(* CoDeSys 2.3.9.42 project: komp.pro *)
(* Libraries: Standard.lib 2.12.10 17:48:34, SYSLIBCALLBACK.LIB 2.12.10 17:48:32 *)

(* PLC configuration (modules and I/O channels)
0750-1405 16 DI 24V DC 3.0ms [Type_1_16_Channels] node 0, in %IB24 out %QB0 {INTTypePAAssignment = PLC; INTTypeModule = plugged}
  AT %IX12.0 [BOOLOnX_I] Ch_1 Digital input
  AT %IX12.1 [BOOLOnX_I] Ch_2 Digital input
  AT %IX12.2 [BOOLOnX_I] Ch_3 Digital input
  AT %IX12.3 [BOOLOnX_I] Ch_4 Digital input
  AT %IX12.4 [BOOLOnX_I] Ch_5 Digital input
  AT %IX12.5 [BOOLOnX_I] Ch_6 Digital input
  AT %IX12.6 [BOOLOnX_I] Ch_7 Digital input
  AT %IX12.7 [BOOLOnX_I] Ch_8 Digital input
  AT %IX12.8 [BOOLOnX_I] Ch_9 Digital input
  AT %IX12.9 [BOOLOnX_I] Ch_10 Digital input
  AT %IX12.10 [BOOLOnX_I] Ch_11 Digital input
  AT %IX12.11 [BOOLOnX_I] Ch_12 Digital input
  AT %IX12.12 [BOOLOnX_I] Ch_13 Digital input
  AT %IX12.13 [BOOLOnX_I] Ch_14 Digital input
  AT %IX12.14 [BOOLOnX_I] Ch_15 Digital input
  AT %IX12.15 [BOOLOnX_I] Ch_16 Digital input
0750-1405 16 DI 24V DC 3.0ms [Type_1_16_Channels] node 0, in %IB24 out %QB0 {INTTypePAAssignment = PLC; INTTypeModule = plugged}
  AT %IX13.0 [BOOLOnX_I] Ch_1 Digital input
  AT %IX13.1 [BOOLOnX_I] Ch_2 Digital input
  AT %IX13.2 [BOOLOnX_I] Ch_3 Digital input
  AT %IX13.3 [BOOLOnX_I] Ch_4 Digital input
  AT %IX13.4 [BOOLOnX_I] Ch_5 Digital input
  AT %IX13.5 [BOOLOnX_I] Ch_6 Digital input
  AT %IX13.6 [BOOLOnX_I] Ch_7 Digital input
  AT %IX13.7 [BOOLOnX_I] Ch_8 Digital input
  AT %IX13.8 [BOOLOnX_I] Ch_9 Digital input
  AT %IX13.9 [BOOLOnX_I] Ch_10 Digital input
  AT %IX13.10 [BOOLOnX_I] Ch_11 Digital input
  AT %IX13.11 [BOOLOnX_I] Ch_12 Digital input
  AT %IX13.12 [BOOLOnX_I] Ch_13 Digital input
  AT %IX13.13 [BOOLOnX_I] Ch_14 Digital input
  AT %IX13.14 [BOOLOnX_I] Ch_15 Digital input
  AT %IX13.15 [BOOLOnX_I] Ch_16 Digital input
0750-1505 16 DO 24V DC 0.5A / LSS [Type_10_16_Channels] node 2, in %IB26 out %QB0 {INTTypePAAssignment = PLC; INTTypeModule = plugged}
  AT %QX0.0 [BOOLOnX_Q] Ch_1 Digital output
  AT %QX0.1 [BOOLOnX_Q] Ch_2 Digital output
  AT %QX0.2 [BOOLOnX_Q] Ch_3 Digital output
  AT %QX0.3 [BOOLOnX_Q] Ch_4 Digital output
  AT %QX0.4 [BOOLOnX_Q] Ch_5 Digital output
  AT %QX0.5 [BOOLOnX_Q] Ch_6 Digital output
  AT %QX0.6 [BOOLOnX_Q] Ch_7 Digital output
  AT %QX0.7 [BOOLOnX_Q] Ch_8 Digital output
  AT %QX0.8 [BOOLOnX_Q] Ch_9 Digital output
  AT %QX0.9 [BOOLOnX_Q] Ch_10 Digital output
  AT %QX0.10 [BOOLOnX_Q] Ch_11 Digital output
  AT %QX0.11 [BOOLOnX_Q] Ch_12 Digital output
  AT %QX0.12 [BOOLOnX_Q] Ch_13 Digital output
  AT %QX0.13 [BOOLOnX_Q] Ch_14 Digital output
  AT %QX0.14 [BOOLOnX_Q] Ch_15 Digital output
  AT %QX0.15 [BOOLOnX_Q] Ch_16 Digital output
0750-1505 16 DO 24V DC 0.5A / LSS [Type_10_16_Channels] node 3, in %IB28 out %QB0 {INTTypePAAssignment = PLC; INTTypeModule = plugged}
  AT %QX1.0 [BOOLOnX_Q] Ch_1 Digital output
  AT %QX1.1 [BOOLOnX_Q] Ch_2 Digital output
  AT %QX1.2 [BOOLOnX_Q] Ch_3 Digital output
  AT %QX1.3 [BOOLOnX_Q] Ch_4 Digital output
  AT %QX1.4 [BOOLOnX_Q] Ch_5 Digital output
  AT %QX1.5 [BOOLOnX_Q] Ch_6 Digital output
  AT %QX1.6 [BOOLOnX_Q] Ch_7 Digital output
  AT %QX1.7 [BOOLOnX_Q] Ch_8 Digital output
  AT %QX1.8 [BOOLOnX_Q] Ch_9 Digital output
  AT %QX1.9 [BOOLOnX_Q] Ch_10 Digital output
  AT %QX1.10 [BOOLOnX_Q] Ch_11 Digital output
  AT %QX1.11 [BOOLOnX_Q] Ch_12 Digital output
  AT %QX1.12 [BOOLOnX_Q] Ch_13 Digital output
  AT %QX1.13 [BOOLOnX_Q] Ch_14 Digital output
  AT %QX1.14 [BOOLOnX_Q] Ch_15 Digital output
  AT %QX1.15 [BOOLOnX_Q] Ch_16 Digital output
0750-0610 24V DC Power Supply / Fuse / Diagn. [Type_1_2_Channels] node 4, in %IB28 out %QB2 {INTTypePAAssignment = PLC; INTTypeModule = plugged}
  AT %IX14.0 [BOOLOnX_I] Ch_1 Digital input
  AT %IX14.1 [BOOLOnX_I] Ch_2 Digital input
0753-0455 4 AI 4-20mA s.e. [Type_8_4_Channels] node 5, in %IB16 out %QB0 {INTTypePAAssignment = PLC; INTTypeModule = plugged}
  AT %IW0 [WORDOnW_I] Ch_1 Input word
  AT %IW1 [WORDOnW_I] Ch_2 Input word
  AT %IW2 [WORDOnW_I] Ch_3 Input word
  AT %IW3 [WORDOnW_I] Ch_4 Input word
0753-0455 4 AI 4-20mA s.e. [Type_8_4_Channels] node 6, in %IB16 out %QB0 {INTTypePAAssignment = PLC; INTTypeModule = plugged}
  AT %IW4 [WORDOnW_I] Ch_1 Input word
  AT %IW5 [WORDOnW_I] Ch_2 Input word
  AT %IW6 [WORDOnW_I] Ch_3 Input word
  AT %IW7 [WORDOnW_I] Ch_4 Input word
0753-0455 4 AI 4-20mA s.e. [Type_8_4_Channels] node 7, in %IB24 out %QB0 {INTTypePAAssignment = PLC; INTTypeModule = plugged}
  AT %IW8 [WORDOnW_I] Ch_1 Input word
  AT %IW9 [WORDOnW_I] Ch_2 Input word
  AT %IW10 [WORDOnW_I] Ch_3 Input word
  AT %IW11 [WORDOnW_I] Ch_4 Input word
AT %IX14.2 [BOOLOnX_I] Ch_1 Digital input
AT %QX2.0 [BOOLOnX_Q] Ch_1 Digital output
AT %IX14.3 [BOOLOnX_I] Ch_2 Digital input
AT %QX2.1 [BOOLOnX_Q] Ch_2 Digital output
AT %IX14.4 [BOOLOnX_I] Ch_3 Digital input
AT %QX2.2 [BOOLOnX_Q] Ch_3 Digital output
AT %IX14.5 [BOOLOnX_I] Ch_4 Digital input
AT %QX2.3 [BOOLOnX_Q] Ch_4 Digital output
AT %IX14.6 [BOOLOnX_I] Ch_5 Digital input
AT %QX2.4 [BOOLOnX_Q] Ch_5 Digital output
AT %IX14.7 [BOOLOnX_I] Ch_6 Digital input
AT %QX2.5 [BOOLOnX_Q] Ch_6 Digital output
AT %IX14.8 [BOOLOnX_I] Ch_7 Digital input
AT %QX2.6 [BOOLOnX_Q] Ch_7 Digital output
AT %IX14.9 [BOOLOnX_I] Ch_8 Digital input
AT %QX2.7 [BOOLOnX_Q] Ch_8 Digital output
0750-1405 16 DI 24V DC 3.0ms [Type_1_16_Channels] node 1, in %IX14.2 out %QB4 {INTTypePAAssignment = PLC; INTTypeModule = plugged}
  AT %IX14.10 [BOOLOnX_I] Ch_1 Digital input
  AT %IX14.11 [BOOLOnX_I] Ch_2 Digital input
  AT %IX14.12 [BOOLOnX_I] Ch_3 Digital input
  AT %IX14.13 [BOOLOnX_I] Ch_4 Digital input
  AT %IX14.14 [BOOLOnX_I] Ch_5 Digital input
  AT %IX14.15 [BOOLOnX_I] Ch_6 Digital input
  AT %IX15.0 [BOOLOnX_I] Ch_7 Digital input
  AT %IX15.1 [BOOLOnX_I] Ch_8 Digital input
  AT %IX15.2 [BOOLOnX_I] Ch_9 Digital input
  AT %IX15.3 [BOOLOnX_I] Ch_10 Digital input
  AT %IX15.4 [BOOLOnX_I] Ch_11 Digital input
  AT %IX15.5 [BOOLOnX_I] Ch_12 Digital input
  AT %IX15.6 [BOOLOnX_I] Ch_13 Digital input
  AT %IX15.7 [BOOLOnX_I] Ch_14 Digital input
  AT %IX15.8 [BOOLOnX_I] Ch_15 Digital input
  AT %IX15.9 [BOOLOnX_I] Ch_16 Digital input
Fieldbus variables [FB_VARS] node 1, in %IB0 out %QB0
Flag variables [FLAG_VARS] node 2, in %IB0 out %QB0
*)

(* Global variable list: Global_Variables *)
VAR_GLOBAL
	waterPump1 : Pumps;
	waterPump2 : Pumps;
	oilPump1 : Pumps;
	oilPump2 : Pumps;
	_18gate : GateValve;
	_4gate : GateValve;
	_5gate : GateValve;
	_6gate : GateValve;
	_7gate : GateValve;
	_8gate : GateValve;
	_9gate : GateValve;
	_10gate : GateValve;
	_11gate : GateValve;
	_14gate : GateValve;
	_17gate : GateValve;
	_19gate : GateValve;
	_20gate : GateValve;
	heater : Heaters;
	komp : Compressor;

	wtrTimeWORD AT %QW256: WORD := 2;
	oilTimeWORD  AT %QW257: WORD := 2;

	MODE AT %QW280 : WORD;

	gate18TimeWORD  AT %IW258 :WORD := 2;
	gate4TimeWORD  AT %IW259 :WORD := 2;
	gate5TimeWORD  AT %IW260 :WORD := 2;
	gate6TimeWORD  AT %IW261 :WORD := 2;
	gate7TimeWORD  AT %IW262 :WORD := 2;
	gate8TimeWORD  AT %IW263 :WORD := 2;
	gate9TimeWORD  AT %IW264 :WORD := 2;
	gate10TimeWORD  AT %IW265 :WORD := 2;
	gate11TimeWORD  AT %IW266 :WORD := 2;
	gate14TimeWORD  AT %IW267 :WORD := 2;
	gate17TimeWORD  AT %QW268 :WORD := 2;
	gate17T3  AT %IW268 :WORD := 3;
	gate17T4  AT %MW268 :WORD := 4;
	wtrTime : TIME := T#2s;
	oilTime : TIME := T#2s;
	gate18Time  :TIME := T#2s;
	gate4Time  :TIME := T#2s;
	gate5Time  :TIME := T#2s;
	gate6Time  :TIME := T#2s;
	gate7Time  :TIME := T#2s;
	gate8Time  :TIME := T#2s;
	gate9Time  :TIME := T#2s;
	gate10Time :TIME := T#2s;
	gate11Time  :TIME := T#2s;
	gate14Time  :TIME := T#2s;
	gate17Time  :TIME := T#2s;

	goRejim AT %QX269.0 : BOOL;
	goPusk AT %QX269.1: BOOL;
	goSTOP AT %QX269.2 : BOOL;
	kompReady AT %QX269.3 : BOOL := FALSE;
	isOK AT %QX269.4: BOOL := TRUE;

	_4gate_open  AT %IX269.5 : BOOL;
	_4gate_close  AT %IX269.6 : BOOL;
	_5gate_open  AT %IX269.7 : BOOL;
	_5gate_close  AT %IX269.8 : BOOL;
	_6gate_open  AT %IX269.9 : BOOL;
	_6gate_close  AT %IX269.10 : BOOL;
	_7gate_open  AT %IX269.11 : BOOL;
	_7gate_close  AT %IX269.12 : BOOL;
	_8gate_open  AT %IX269.13 : BOOL;
	_8gate_close  AT %IX269.14 : BOOL;
	_9gate_open  AT %IX269.15 : BOOL;
	_9gate_close  AT %IX270.0 : BOOL;
	_10gate_open  AT %IX270.1 : BOOL;
	_10gate_close  AT %IX270.2 : BOOL;
	_11gate_open  AT %IX270.3 : BOOL;
	_11gate_close  AT %IX270.4 : BOOL;
	_14gate_open  AT %IX270.5 : BOOL;
	_14gate_close  AT %IX270.6 : BOOL;
	_18gate_open  AT %IX270.7 : BOOL;
	_18gate_close  AT %IX270.8 : BOOL;
	_19gate_open  AT %IX270.9 : BOOL;
	_19gate_close  AT %IX270.10 : BOOL;
	_20gate_open  AT %IX270.11 : BOOL;
	_20gate_close  AT %IX270.12 : BOOL;
	oilPump1_run  AT %IX270.13 : BOOL;
	oilPump2_run  AT %IX270.14 : BOOL;
	waterPump1_run  AT %IX270.15 : BOOL;
	waterPump2_run  AT %IX271.0 : BOOL;
	komp_run  AT %IX271.1 : BOOL;
	komp_stop  AT %IX271.2 : BOOL;
	autoManual  AT %IX272.0 : BOOL;


END_VAR

(* Data type *)
TYPE Compressor :
STRUCT
	run: BOOL;
	stop : BOOL;
	status : BOOL;
END_STRUCT
END_TYPE

(* Data type *)
TYPE GateValve :
STRUCT
	opened: BOOL;
	closed : BOOL;
	open : BOOL;
	close : BOOL;
END_STRUCT
END_TYPE

(* Data type *)
TYPE Heaters :
STRUCT
	status : BOOL;
	run : BOOL;
END_STRUCT
END_TYPE

(* Data type *)
TYPE Pumps :
STRUCT
	status : BOOL;
	run : BOOL;
END_STRUCT
END_TYPE

(* POU PLC_PRG, ST *)
PROGRAM PLC_PRG
VAR
	a : BOOL;
END_VAR
translate();



(*
CASE MODE OF
	10: stop();
	1 : preparation();
END_CASE;




gateManage();

pusk();
stopp();
**)
rejim();
IF(isOK = FALSE) THEN
	goSTOP := TRUE;
END_IF;
END_PROGRAM

(* POU translate, ST *)
PROGRAM translate
VAR

END_VAR
(******************************  M1 ******************************
oilPump.status :=%IX12.0;
waterPump.status := %IX12.1;
_18gate.opened := %IX12.2;
_18gate.closed := %IX12.3;
_4gate.opened := %IX12.4;
_4gate.closed := %IX12.5;
_5gate.opened := %IX12.6;
_5gate.closed := %IX12.7;
_6gate.opened := %IX12.8;
_6gate.closed := %IX12.9;
_7gate.opened := %IX12.10;
_7gate.closed := %IX12.11;
_8gate.opened := %IX12.12;
_8gate.closed := %IX12.13;
_9gate.opened := %IX12.14;
_9gate.closed := %IX12.15;
(*******************************  M1 ******************************)
(******************************  M2 ******************************)
_10gate.opened := %IX13.0;
_10gate.closed := %IX13.1;
_11gate.opened := %IX13.2;
_11gate.opened := %IX13.3;
_14gate.opened := %IX13.4;
_14gate.closed := %IX13.5;
_17gate.opened := %IX13.6;
_17gate.closed := %IX13.7;
heater.status := %IX13.8;
(*******************************  M2 *****************************)
*)
IF (%IX272.0 <> %QX272.0) THEN
	%QX272.0 := %IX272.0;
END_IF;
IF (%QW273 <> %IW273) THEN
		%QW273 := %IW273;
	END_IF;
IF (autoManual = FALSE) THEN
	%QX0.0 := _4gate_open;
	%QX0.1 := _4gate_close;
	%QX0.2 := _5gate_open;;
	%QX0.3 := _5gate_close;
	%QX0.4 := _6gate_open;
	%QX0.5 := _6gate_close;
	%QX0.6 := _7gate_open;
	%QX0.7 := _7gate_close;
	%QX0.8 := _8gate_open;
	%QX0.9 := _8gate_close;
	%QX0.10 := _9gate_open;
	%QX0.11 := _9gate_close;
	%QX0.12 := _10gate_open;
	%QX0.13 := _10gate_close;
	%QX0.14 := _11gate_open;
	%QX0.15 := _11gate_close;
	%QX1.0 := _14gate_open;
	%QX1.1 := _14gate_close;
	%QX1.2 := _18gate_open;
	%QX1.3 := _18gate_close;
	%QX1.4 := _19gate_open;
	%QX1.5 := _19gate_close;
	%QX1.6 := _20gate_open;
	%QX1.7 := _20gate_close;
	%QX1.8 := oilPump1_run;
	%QX1.9 := oilPump2.run;
	%QX1.10 := waterPump1_run;
	%QX1.11 := waterPump2_run;
	%QX1.12 := komp_run;
	%QX1.13 := komp_stop;
	%QX1.14 := goRejim;
	%QX1.15 := goPusk;
	IF (%QW269 <> %IW269) THEN
		%QW269 := %IW269;
	END_IF;
	IF (%QW270 <> %IW270) THEN
		%QW270 := %IW270;
	END_IF;
	IF (%QW271 <> %IW271) THEN
		%QW271 := %IW271;
	END_IF;
ELSE
	%QX0.0 := _4gate.open;
	%QX0.1 := _4gate.close;
	%QX0.2 := _5gate.open;;
	%QX0.3 := _5gate.close;
	%QX0.4 := _6gate.open;
	%QX0.5 := _6gate.close;
	%QX0.6 := _7gate.open;
	%QX0.7 := _7gate.close;
	%QX0.8 := _8gate.open;
	%QX0.9 := _8gate.close;
	%QX0.10 := _9gate.open;
	%QX0.11 := _9gate.close;
	%QX0.12 := _10gate.open;
	%QX0.13 := _10gate.close;
	%QX0.14 := _11gate.open;
	%QX0.15 := _11gate.close;
	%QX1.0 := _14gate.open;
	%QX1.1 := _14gate.close;
	%QX1.2 := _18gate.open;
	%QX1.3 := _18gate.close;
	%QX1.4 := _19gate.open;
	%QX1.5 := _19gate.close;
	%QX1.6 := _20gate.open;
	%QX1.7 := _20gate.close;
	%QX1.8 := oilPump1.run;
	%QX1.9 := oilPump2.run;
	%QX1.10 := waterPump1.run;
	%QX1.11 := waterPump2.run;
	%QX1.12 := komp.run;
	%QX1.13 := komp.stop;
	%QX1.14 := goRejim;
	%QX1.15 := goPusk;

END_IF;

(*******************************  M3  ******************************)
(*******************************  TIME  ******************************)
wtrTime := T#1s * wtrTimeWORD;
oilTime := T#1s* oilTimeWORD;
gate18Time := T#1s * gate18TimeWORD;
gate4Time := T#1s * gate4TimeWORD;
gate5Time := T#1s * gate5TimeWORD;
gate6Time := T#1s * gate6TimeWORD;
gate7Time := T#1s * gate7TimeWORD;
gate8Time := T#1s * gate8TimeWORD;
gate9Time :=  T#1s * gate9TimeWORD;
gate10Time := T#1s * gate10TimeWORD;
gate11Time := T#1s * gate11TimeWORD;
gate14Time := T#1s * gate14TimeWORD;
gate17Time := T#1s * gate17TimeWORD;
(*******************************  TIME  ******************************)
(*******************************  TIME  ******************************)
END_PROGRAM

(* POU stop, CFC *)
PROGRAM stop
VAR
END_VAR
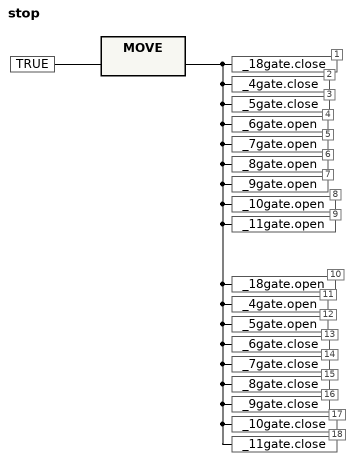
_CFC_ (* Continuous Function Chart, elements in execution order *)
#0 MOVE(TRUE)
#1 _18gate.close <= #0
#2 _4gate.close <= #0
#3 _5gate.close <= #0
#4 _6gate.open <= #0
#5 _7gate.open <= #0
#6 _8gate.open <= #0
#7 _9gate.open <= #0
#8 _10gate.open <= #0
#9 _11gate.open <= #0
#10 _18gate.open <= #0
#11 _4gate.open <= #0
#12 _5gate.open <= #0
#13 _6gate.close <= #0
#14 _7gate.close <= #0
#15 _8gate.close <= #0
#16 _9gate.close <= #0
#17 _10gate.close <= #0
#18 _11gate.close <= #0
_END_CFC_
(* the same logic as Structured Text *)
_18gate.close := TRUE;
_4gate.close := TRUE;
_5gate.close := TRUE;
_6gate.open := TRUE;
_7gate.open := TRUE;
_8gate.open := TRUE;
_9gate.open := TRUE;
_10gate.open := TRUE;
_11gate.open := TRUE;
_18gate.open := TRUE;
_4gate.open := TRUE;
_5gate.open := TRUE;
_6gate.close := TRUE;
_7gate.close := TRUE;
_8gate.close := TRUE;
_9gate.close := TRUE;
_10gate.close := TRUE;
_11gate.close := TRUE;
END_PROGRAM

(* POU rejim, LD *)
PROGRAM rejim
VAR
	waterTON: TON;
	oilTON: TON;
	gate18TON: TON;
	gate4TON: TON;
	gate14TON: TON;
	gate11TON: TON;
	kompTON: TON;
	kompTOF: TOF;
	kompTP: TP;
	kompTRIGF: F_TRIG;
	kompTEMP : BOOL;
END_VAR
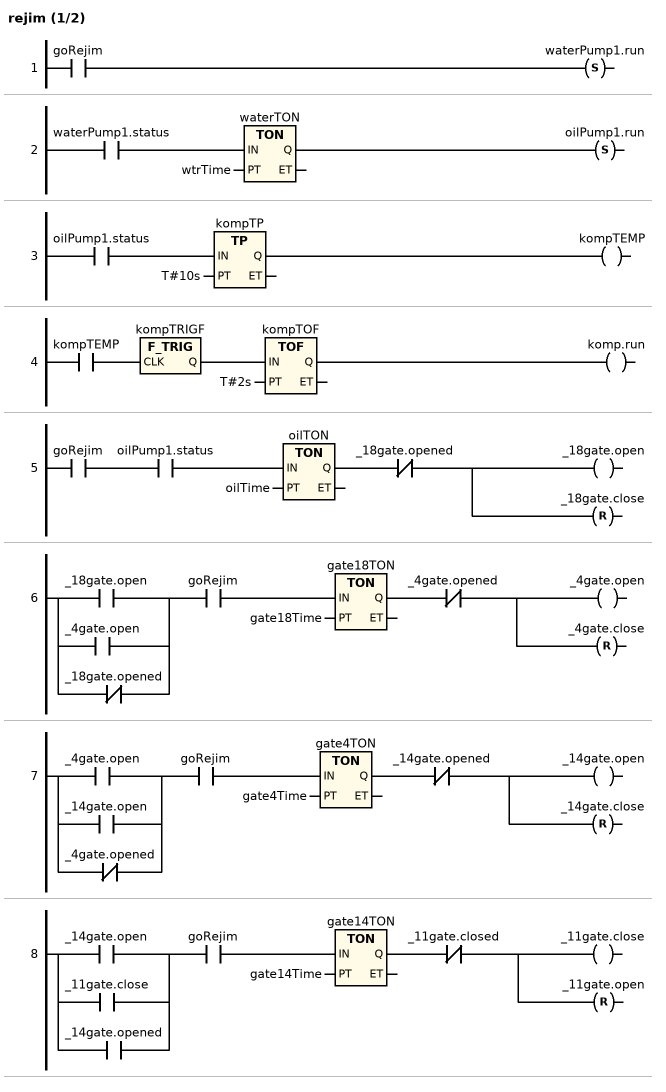
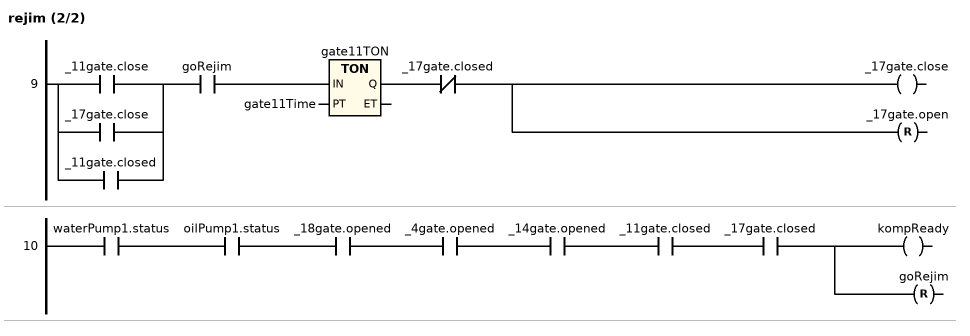
_LD_ (* Ladder Diagram *)
NETWORK 1
	[goRejim] --- (S waterPump1.run)
NETWORK 2
	[waterPump1.status] - waterTON:TON(IN: *, PT: wtrTime) --- (S oilPump1.run)
NETWORK 3
	[oilPump1.status] - kompTP:TP(IN: *, PT: T#10s) --- (kompTEMP)
NETWORK 4
	[kompTEMP] - kompTRIGF:F_TRIG(CLK: *) - kompTOF:TOF(IN: *, PT: T#2s) --- (komp.run)
NETWORK 5
	[goRejim] - [oilPump1.status] - oilTON:TON(IN: *, PT: oilTime) - [/_18gate.opened] --- (_18gate.open) (R _18gate.close)
NETWORK 6
	{ [_18gate.open] | [_4gate.open] | [/_18gate.opened] } - [goRejim] - gate18TON:TON(IN: *, PT: gate18Time) - [/_4gate.opened] --- (_4gate.open) (R _4gate.close)
NETWORK 7
	{ [_4gate.open] | [_14gate.open] | [/_4gate.opened] } - [goRejim] - gate4TON:TON(IN: *, PT: gate4Time) - [/_14gate.opened] --- (_14gate.open) (R _14gate.close)
NETWORK 8
	{ [_14gate.open] | [_11gate.close] | [_14gate.opened] } - [goRejim] - gate14TON:TON(IN: *, PT: gate14Time) - [/_11gate.closed] --- (_11gate.close) (R _11gate.open)
NETWORK 9
	{ [_11gate.close] | [_17gate.close] | [_11gate.closed] } - [goRejim] - gate11TON:TON(IN: *, PT: gate11Time) - [/_17gate.closed] --- (_17gate.close) (R _17gate.open)
NETWORK 10
	[waterPump1.status] - [oilPump1.status] - [_18gate.opened] - [_4gate.opened] - [_14gate.opened] - [_11gate.closed] - [_17gate.closed] --- (kompReady) (R goRejim)
_END_LD_
(* the same logic as Structured Text *)
(* Network 1 *)
IF goRejim THEN waterPump1.run := TRUE; END_IF;
(* Network 2 *)
waterTON(IN := waterPump1.status, PT := wtrTime);
IF waterTON.Q THEN oilPump1.run := TRUE; END_IF;
(* Network 3 *)
kompTP(IN := oilPump1.status, PT := T#10s);
kompTEMP := kompTP.Q;
(* Network 4 *)
kompTRIGF(CLK := kompTEMP);
kompTOF(IN := kompTRIGF.Q, PT := T#2s);
komp.run := kompTOF.Q;
(* Network 5 *)
oilTON(IN := goRejim AND oilPump1.status, PT := oilTime);
_18gate.open := oilTON.Q AND NOT _18gate.opened;
IF _18gate.open THEN _18gate.close := FALSE; END_IF;
(* Network 6 *)
gate18TON(IN := (_18gate.open OR _4gate.open OR NOT _18gate.opened) AND goRejim, PT := gate18Time);
_4gate.open := gate18TON.Q AND NOT _4gate.opened;
IF _4gate.open THEN _4gate.close := FALSE; END_IF;
(* Network 7 *)
gate4TON(IN := (_4gate.open OR _14gate.open OR NOT _4gate.opened) AND goRejim, PT := gate4Time);
_14gate.open := gate4TON.Q AND NOT _14gate.opened;
IF _14gate.open THEN _14gate.close := FALSE; END_IF;
(* Network 8 *)
gate14TON(IN := (_14gate.open OR _11gate.close OR _14gate.opened) AND goRejim, PT := gate14Time);
_11gate.close := gate14TON.Q AND NOT _11gate.closed;
IF _11gate.close THEN _11gate.open := FALSE; END_IF;
(* Network 9 *)
gate11TON(IN := (_11gate.close OR _17gate.close OR _11gate.closed) AND goRejim, PT := gate11Time);
_17gate.close := gate11TON.Q AND NOT _17gate.closed;
IF _17gate.close THEN _17gate.open := FALSE; END_IF;
(* Network 10 *)
kompReady := waterPump1.status AND oilPump1.status AND _18gate.opened AND _4gate.opened AND _14gate.opened AND _11gate.closed AND _17gate.closed;
IF kompReady THEN goRejim := FALSE; END_IF;
END_PROGRAM

(* POU LAB/gateManage, CFC *)
PROGRAM gateManage
VAR
	gate18 : fbGateManage;
	gate4: fbGateManage;
	gate11: fbGateManage;
	gate17: fbGateManage;
	gate14: fbGateManage;
	gate5: fbGateManage;
	gate8: fbGateManage;
	gate7: fbGateManage;
	gate9: fbGateManage;
	gate10: fbGateManage;
	gate6: fbGateManage;
	wtrPump: fbPumpManage;
	olPump: fbPumpManage;
END_VAR
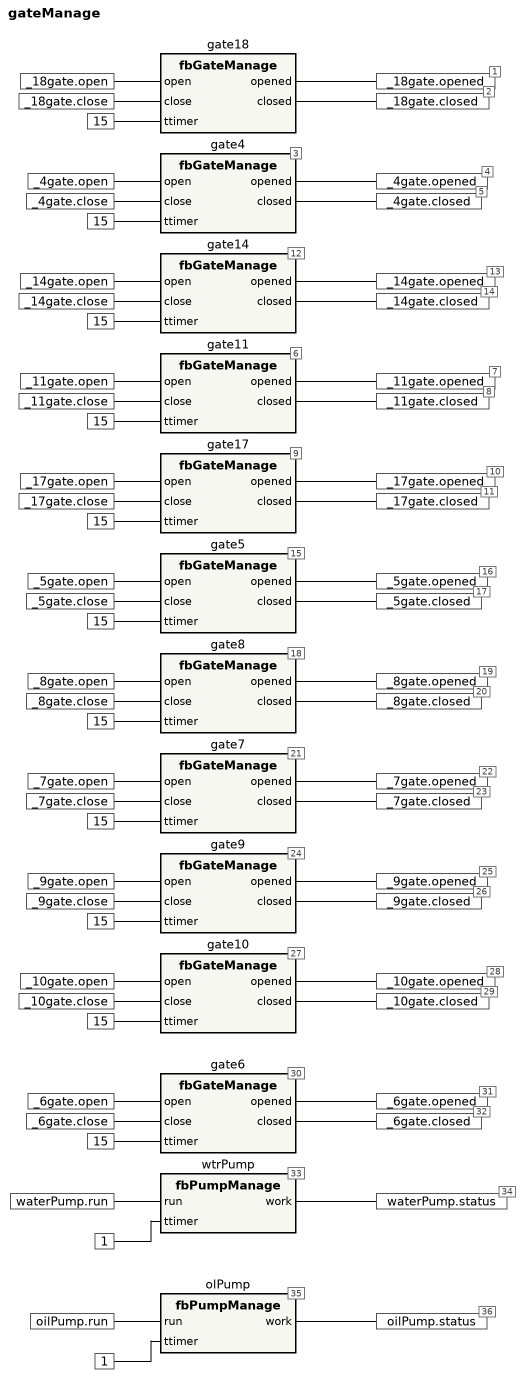
_CFC_ (* Continuous Function Chart, elements in execution order *)
#0 gate18:fbGateManage(open: _18gate.open, close: _18gate.close, ttimer: 15)
#1 _18gate.opened <= #0.opened
#2 _18gate.closed <= #0.closed
#3 gate4:fbGateManage(open: _4gate.open, close: _4gate.close, ttimer: 15)
#4 _4gate.opened <= #3.opened
#5 _4gate.closed <= #3.closed
#6 gate11:fbGateManage(open: _11gate.open, close: _11gate.close, ttimer: 15)
#7 _11gate.opened <= #6.opened
#8 _11gate.closed <= #6.closed
#9 gate17:fbGateManage(open: _17gate.open, close: _17gate.close, ttimer: 15)
#10 _17gate.opened <= #9.opened
#11 _17gate.closed <= #9.closed
#12 gate14:fbGateManage(open: _14gate.open, close: _14gate.close, ttimer: 15)
#13 _14gate.opened <= #12.opened
#14 _14gate.closed <= #12.closed
#15 gate5:fbGateManage(open: _5gate.open, close: _5gate.close, ttimer: 15)
#16 _5gate.opened <= #15.opened
#17 _5gate.closed <= #15.closed
#18 gate8:fbGateManage(open: _8gate.open, close: _8gate.close, ttimer: 15)
#19 _8gate.opened <= #18.opened
#20 _8gate.closed <= #18.closed
#21 gate7:fbGateManage(open: _7gate.open, close: _7gate.close, ttimer: 15)
#22 _7gate.opened <= #21.opened
#23 _7gate.closed <= #21.closed
#24 gate9:fbGateManage(open: _9gate.open, close: _9gate.close, ttimer: 15)
#25 _9gate.opened <= #24.opened
#26 _9gate.closed <= #24.closed
#27 gate10:fbGateManage(open: _10gate.open, close: _10gate.close, ttimer: 15)
#28 _10gate.opened <= #27.opened
#29 _10gate.closed <= #27.closed
#30 gate6:fbGateManage(open: _6gate.open, close: _6gate.close, ttimer: 15)
#31 _6gate.opened <= #30.opened
#32 _6gate.closed <= #30.closed
#33 wtrPump:fbPumpManage(run: waterPump.run, ttimer: 1)
#34 waterPump.status <= #33.work
#35 olPump:fbPumpManage(run: oilPump.run, ttimer: 1)
#36 oilPump.status <= #35.work
_END_CFC_
(* the same logic as Structured Text *)
gate18(open := _18gate.open, close := _18gate.close, ttimer := 15);
_18gate.opened := gate18.opened;
_18gate.closed := gate18.closed;
gate4(open := _4gate.open, close := _4gate.close, ttimer := 15);
_4gate.opened := gate4.opened;
_4gate.closed := gate4.closed;
gate11(open := _11gate.open, close := _11gate.close, ttimer := 15);
_11gate.opened := gate11.opened;
_11gate.closed := gate11.closed;
gate17(open := _17gate.open, close := _17gate.close, ttimer := 15);
_17gate.opened := gate17.opened;
_17gate.closed := gate17.closed;
gate14(open := _14gate.open, close := _14gate.close, ttimer := 15);
_14gate.opened := gate14.opened;
_14gate.closed := gate14.closed;
gate5(open := _5gate.open, close := _5gate.close, ttimer := 15);
_5gate.opened := gate5.opened;
_5gate.closed := gate5.closed;
gate8(open := _8gate.open, close := _8gate.close, ttimer := 15);
_8gate.opened := gate8.opened;
_8gate.closed := gate8.closed;
gate7(open := _7gate.open, close := _7gate.close, ttimer := 15);
_7gate.opened := gate7.opened;
_7gate.closed := gate7.closed;
gate9(open := _9gate.open, close := _9gate.close, ttimer := 15);
_9gate.opened := gate9.opened;
_9gate.closed := gate9.closed;
gate10(open := _10gate.open, close := _10gate.close, ttimer := 15);
_10gate.opened := gate10.opened;
_10gate.closed := gate10.closed;
gate6(open := _6gate.open, close := _6gate.close, ttimer := 15);
_6gate.opened := gate6.opened;
_6gate.closed := gate6.closed;
wtrPump(run := waterPump.run, ttimer := 1);
waterPump.status := wtrPump.work;
olPump(run := oilPump.run, ttimer := 1);
oilPump.status := olPump.work;
END_PROGRAM

(* POU LAB/fbGateManage, CFC *)
FUNCTION_BLOCK fbGateManage
VAR_INPUT
	open : BOOL;
	close : BOOL;
	ttimer : WORD;
END_VAR
VAR_OUTPUT
	opened : BOOL;
	closed : BOOL;
END_VAR
VAR
	t :TIME := T#20s;
	tOpen: TON;
	tClose: TON;
	OpenTON : TON;
END_VAR
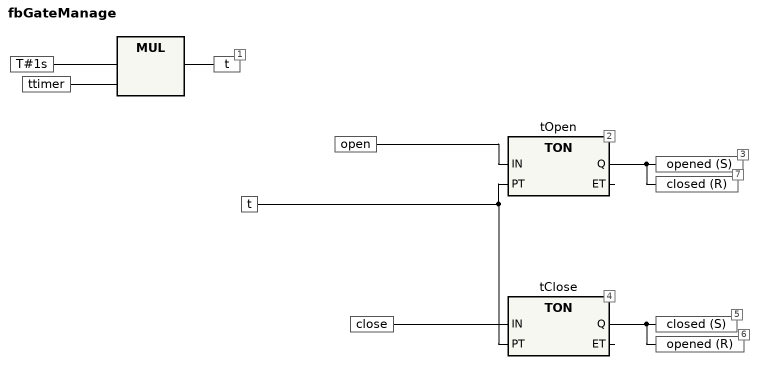
_CFC_ (* Continuous Function Chart, elements in execution order *)
#0 MUL(T#1s, ttimer)
#1 t <= #0
#2 tOpen:TON(IN: open, PT: t)
#3 S opened <= #2.Q
#4 tClose:TON(IN: close, PT: t)
#5 S closed <= #4.Q
#6 R opened <= #4.Q
#7 R closed <= #2.Q
_END_CFC_
(* the same logic as Structured Text *)
t := T#1s * ttimer;
tOpen(IN := open, PT := t);
IF tOpen.Q THEN opened := TRUE; END_IF;
tClose(IN := close, PT := t);
IF tClose.Q THEN closed := TRUE; END_IF;
IF tClose.Q THEN opened := FALSE; END_IF;
IF tOpen.Q THEN closed := FALSE; END_IF;
END_FUNCTION_BLOCK

(* POU LAB/fbPumpManage, CFC *)
FUNCTION_BLOCK fbPumpManage
VAR_INPUT
	run : BOOL;
	ttimer : WORD := 1;
END_VAR
VAR_OUTPUT
	work : BOOL;
END_VAR
VAR
	tOpen: TON;
	tClose: TON;
	trig: F_TRIG;
END_VAR
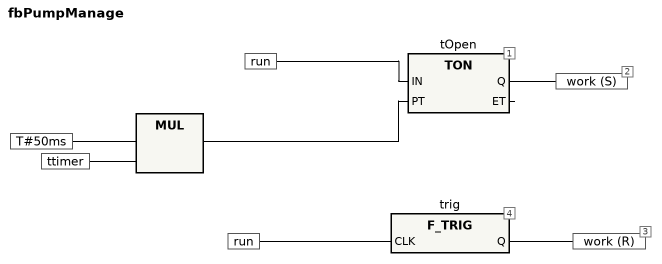
_CFC_ (* Continuous Function Chart, elements in execution order *)
#0 MUL(T#50ms, ttimer)
#1 tOpen:TON(IN: run, PT: #0)
#2 S work <= #1.Q
#3 R work <= #4.Q
#4 trig:F_TRIG(CLK: run)
_END_CFC_
(* the same logic as Structured Text *)
tOpen(IN := run, PT := T#50ms * ttimer);
IF tOpen.Q THEN work := TRUE; END_IF;
IF trig.Q THEN work := FALSE; END_IF;
trig(CLK := run);
END_FUNCTION_BLOCK

(* POU preparation, CFC *)
PROGRAM preparation
VAR
	rswater: RS;
	wtrTime : TIME := T#10s;
	wtrTON :TON;
	go : BOOL := TRUE;

	mmm: WORD;
END_VAR
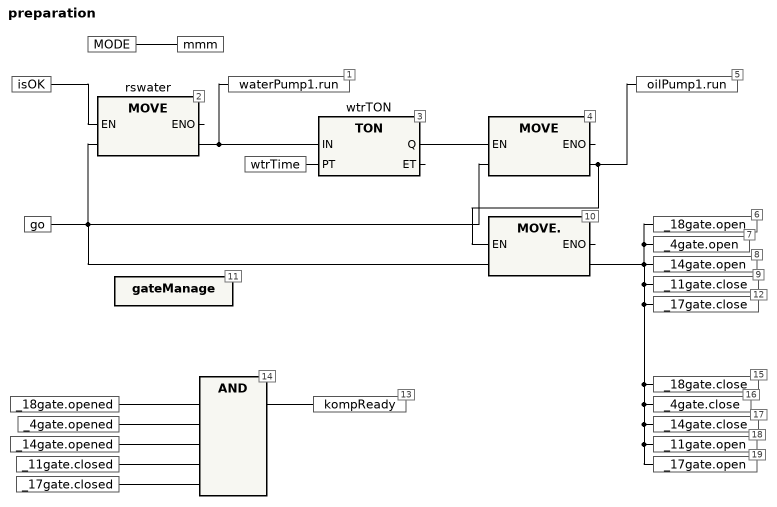
_CFC_ (* Continuous Function Chart, elements in execution order *)
#0 mmm <= MODE
#1 waterPump1.run <= #2
#2 rswater:MOVE(EN: isOK, go)
#3 wtrTON:TON(IN: #2, PT: wtrTime)
#4 MOVE(EN: #3.Q, go)
#5 oilPump1.run <= #4
#6 _18gate.open <= #10
#7 _4gate.open <= #10
#8 _14gate.open <= #10
#9 _11gate.close <= #10
#10 MOVE.(EN: #4, go)
#11 gateManage()
#12 _17gate.close <= #10
#13 kompReady <= #14
#14 AND(_18gate.opened, _4gate.opened, _14gate.opened, _11gate.closed, _17gate.closed)
#15 _18gate.close <= #10
#16 _4gate.close <= #10
#17 _14gate.close <= #10
#18 _11gate.open <= #10
#19 _17gate.open <= #10
_END_CFC_
END_PROGRAM

(* POU pusk, LD *)
PROGRAM pusk
VAR
	gate5TON: TON;
	gate8TON: TON;
	gate7TON: TON;
	gate9TON: TON;
	gate10TON: TON;
END_VAR
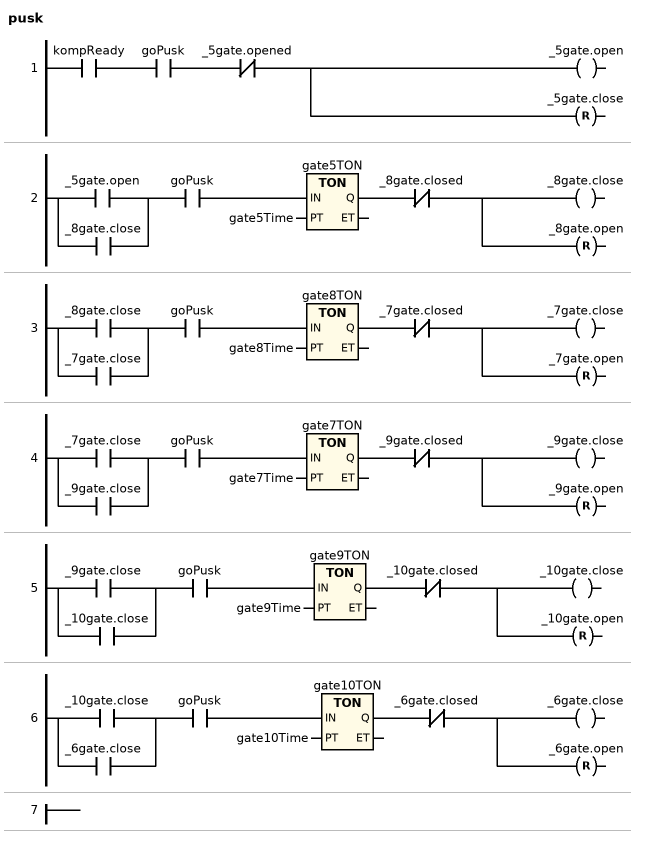
_LD_ (* Ladder Diagram *)
NETWORK 1
	[kompReady] - [goPusk] - [/_5gate.opened] --- (_5gate.open) (R _5gate.close)
NETWORK 2
	{ [_5gate.open] | [_8gate.close] } - [goPusk] - gate5TON:TON(IN: *, PT: gate5Time) - [/_8gate.closed] --- (_8gate.close) (R _8gate.open)
NETWORK 3
	{ [_8gate.close] | [_7gate.close] } - [goPusk] - gate8TON:TON(IN: *, PT: gate8Time) - [/_7gate.closed] --- (_7gate.close) (R _7gate.open)
NETWORK 4
	{ [_7gate.close] | [_9gate.close] } - [goPusk] - gate7TON:TON(IN: *, PT: gate7Time) - [/_9gate.closed] --- (_9gate.close) (R _9gate.open)
NETWORK 5
	{ [_9gate.close] | [_10gate.close] } - [goPusk] - gate9TON:TON(IN: *, PT: gate9Time) - [/_10gate.closed] --- (_10gate.close) (R _10gate.open)
NETWORK 6
	{ [_10gate.close] | [_6gate.close] } - [goPusk] - gate10TON:TON(IN: *, PT: gate10Time) - [/_6gate.closed] --- (_6gate.close) (R _6gate.open)
NETWORK 7
	*
_END_LD_
(* the same logic as Structured Text *)
(* Network 1 *)
_5gate.open := kompReady AND goPusk AND NOT _5gate.opened;
IF _5gate.open THEN _5gate.close := FALSE; END_IF;
(* Network 2 *)
gate5TON(IN := (_5gate.open OR _8gate.close) AND goPusk, PT := gate5Time);
_8gate.close := gate5TON.Q AND NOT _8gate.closed;
IF _8gate.close THEN _8gate.open := FALSE; END_IF;
(* Network 3 *)
gate8TON(IN := (_8gate.close OR _7gate.close) AND goPusk, PT := gate8Time);
_7gate.close := gate8TON.Q AND NOT _7gate.closed;
IF _7gate.close THEN _7gate.open := FALSE; END_IF;
(* Network 4 *)
gate7TON(IN := (_7gate.close OR _9gate.close) AND goPusk, PT := gate7Time);
_9gate.close := gate7TON.Q AND NOT _9gate.closed;
IF _9gate.close THEN _9gate.open := FALSE; END_IF;
(* Network 5 *)
gate9TON(IN := (_9gate.close OR _10gate.close) AND goPusk, PT := gate9Time);
_10gate.close := gate9TON.Q AND NOT _10gate.closed;
IF _10gate.close THEN _10gate.open := FALSE; END_IF;
(* Network 6 *)
gate10TON(IN := (_10gate.close OR _6gate.close) AND goPusk, PT := gate10Time);
_6gate.close := gate10TON.Q AND NOT _6gate.closed;
IF _6gate.close THEN _6gate.open := FALSE; END_IF;
(* Network 7 *)
END_PROGRAM

(* POU stopp, LD *)
PROGRAM stopp
VAR
	trigSTOP: R_TRIG;
	tmp: BOOL;
END_VAR
VAR (* helpers for the ST form of the networks *)
	_p1 : BOOL;
END_VAR
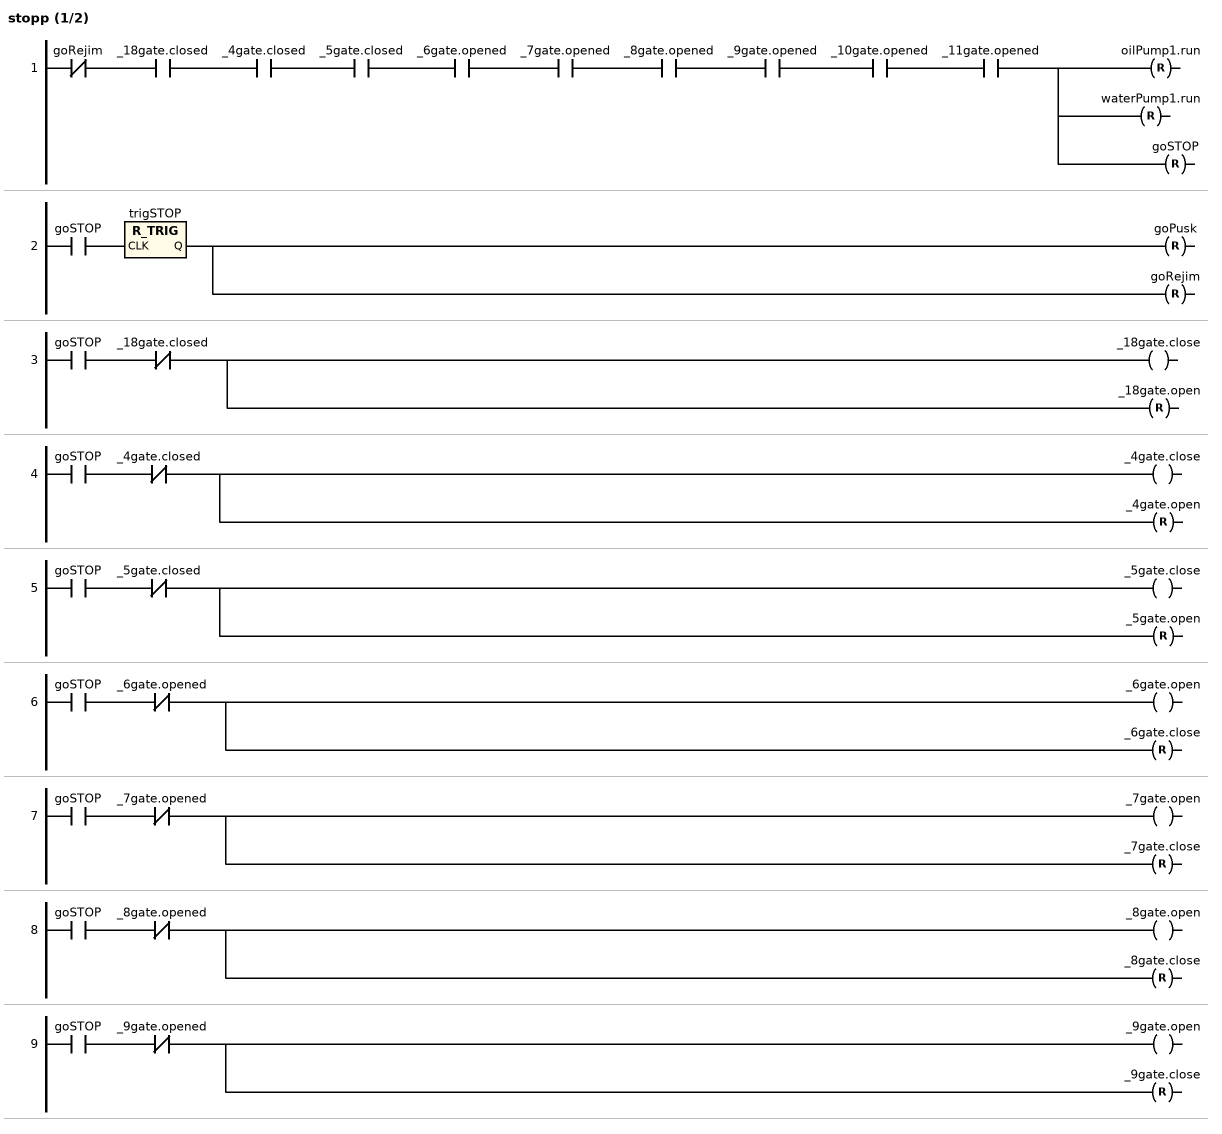
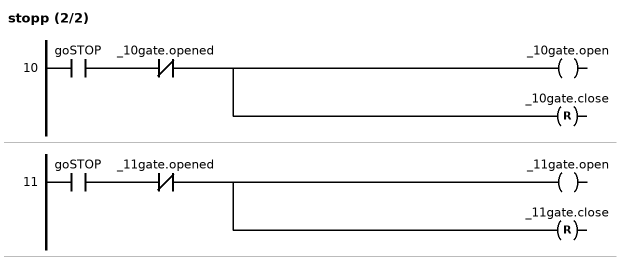
_LD_ (* Ladder Diagram *)
NETWORK 1
	[/goRejim] - [_18gate.closed] - [_4gate.closed] - [_5gate.closed] - [_6gate.opened] - [_7gate.opened] - [_8gate.opened] - [_9gate.opened] - [_10gate.opened] - [_11gate.opened] --- (R oilPump1.run) (R waterPump1.run) (R goSTOP)
NETWORK 2
	[goSTOP] - trigSTOP:R_TRIG(CLK: *) --- (R goPusk) (R goRejim)
NETWORK 3
	[goSTOP] - [/_18gate.closed] --- (_18gate.close) (R _18gate.open)
NETWORK 4
	[goSTOP] - [/_4gate.closed] --- (_4gate.close) (R _4gate.open)
NETWORK 5
	[goSTOP] - [/_5gate.closed] --- (_5gate.close) (R _5gate.open)
NETWORK 6
	[goSTOP] - [/_6gate.opened] --- (_6gate.open) (R _6gate.close)
NETWORK 7
	[goSTOP] - [/_7gate.opened] --- (_7gate.open) (R _7gate.close)
NETWORK 8
	[goSTOP] - [/_8gate.opened] --- (_8gate.open) (R _8gate.close)
NETWORK 9
	[goSTOP] - [/_9gate.opened] --- (_9gate.open) (R _9gate.close)
NETWORK 10
	[goSTOP] - [/_10gate.opened] --- (_10gate.open) (R _10gate.close)
NETWORK 11
	[goSTOP] - [/_11gate.opened] --- (_11gate.open) (R _11gate.close)
_END_LD_
(* the same logic as Structured Text *)
(* Network 1 *)
_p1 := NOT goRejim AND _18gate.closed AND _4gate.closed AND _5gate.closed AND _6gate.opened AND _7gate.opened AND _8gate.opened AND _9gate.opened AND _10gate.opened AND _11gate.opened;
IF _p1 THEN oilPump1.run := FALSE; waterPump1.run := FALSE; goSTOP := FALSE; END_IF;
(* Network 2 *)
trigSTOP(CLK := goSTOP);
IF trigSTOP.Q THEN goPusk := FALSE; goRejim := FALSE; END_IF;
(* Network 3 *)
_18gate.close := goSTOP AND NOT _18gate.closed;
IF _18gate.close THEN _18gate.open := FALSE; END_IF;
(* Network 4 *)
_4gate.close := goSTOP AND NOT _4gate.closed;
IF _4gate.close THEN _4gate.open := FALSE; END_IF;
(* Network 5 *)
_5gate.close := goSTOP AND NOT _5gate.closed;
IF _5gate.close THEN _5gate.open := FALSE; END_IF;
(* Network 6 *)
_6gate.open := goSTOP AND NOT _6gate.opened;
IF _6gate.open THEN _6gate.close := FALSE; END_IF;
(* Network 7 *)
_7gate.open := goSTOP AND NOT _7gate.opened;
IF _7gate.open THEN _7gate.close := FALSE; END_IF;
(* Network 8 *)
_8gate.open := goSTOP AND NOT _8gate.opened;
IF _8gate.open THEN _8gate.close := FALSE; END_IF;
(* Network 9 *)
_9gate.open := goSTOP AND NOT _9gate.opened;
IF _9gate.open THEN _9gate.close := FALSE; END_IF;
(* Network 10 *)
_10gate.open := goSTOP AND NOT _10gate.opened;
IF _10gate.open THEN _10gate.close := FALSE; END_IF;
(* Network 11 *)
_11gate.open := goSTOP AND NOT _11gate.opened;
IF _11gate.open THEN _11gate.close := FALSE; END_IF;
END_PROGRAM

(* Visualisation main
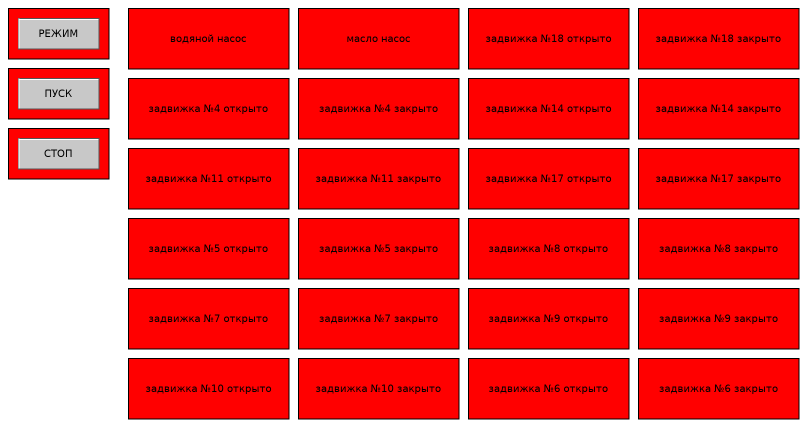
rounded rectangle at (130,10)-(291,71): text "водяной насос"; alarm colour if .waterPump.status
rounded rectangle at (300,10)-(461,71): text "масло насос"; alarm colour if .oilPump.status
rounded rectangle at (470,10)-(631,71): text "задвижка №18 открыто"; alarm colour if ._18gate.opened
rounded rectangle at (640,10)-(801,71): text "задвижка №18 закрыто"; alarm colour if ._18gate.closed
rounded rectangle at (130,80)-(291,141): text "задвижка №4 открыто"; alarm colour if ._4gate.opened
rounded rectangle at (300,80)-(461,141): text "задвижка №4 закрыто"; alarm colour if ._4gate.closed
rounded rectangle at (470,80)-(631,141): text "задвижка №14 открыто"; alarm colour if ._14gate.opened
rounded rectangle at (640,80)-(801,141): text "задвижка №14 закрыто"; alarm colour if ._14gate.closed
rounded rectangle at (130,150)-(291,211): text "задвижка №11 открыто"; alarm colour if ._11gate.opened
rounded rectangle at (300,150)-(461,211): text "задвижка №11 закрыто"; alarm colour if ._11gate.closed
rounded rectangle at (470,150)-(631,211): text "задвижка №17 открыто"; alarm colour if ._17gate.opened
rounded rectangle at (640,150)-(801,211): text "задвижка №17 закрыто"; alarm colour if ._17gate.closed
rounded rectangle at (130,220)-(291,281): text "задвижка №5 открыто"; alarm colour if ._5gate.opened
rounded rectangle at (300,220)-(461,281): text "задвижка №5 закрыто"; alarm colour if ._5gate.closed
rounded rectangle at (470,220)-(631,281): text "задвижка №8 открыто"; alarm colour if ._8gate.opened
rounded rectangle at (640,220)-(801,281): text "задвижка №8 закрыто"; alarm colour if ._8gate.closed
rounded rectangle at (130,290)-(291,351): text "задвижка №7 открыто"; alarm colour if ._7gate.opened
rounded rectangle at (300,290)-(461,351): text "задвижка №7 закрыто"; alarm colour if ._7gate.closed
rounded rectangle at (470,290)-(631,351): text "задвижка №9 открыто"; alarm colour if ._9gate.opened
rounded rectangle at (640,290)-(801,351): text "задвижка №9 закрыто"; alarm colour if ._9gate.closed
rounded rectangle at (130,360)-(291,421): text "задвижка №10 открыто"; alarm colour if ._10gate.opened
rounded rectangle at (300,360)-(461,421): text "задвижка №10 закрыто"; alarm colour if ._10gate.closed
rounded rectangle at (470,360)-(631,421): text "задвижка №6 открыто"; alarm colour if ._6gate.opened
rounded rectangle at (640,360)-(801,421): text "задвижка №6 закрыто"; alarm colour if ._6gate.closed
rounded rectangle at (10,130)-(111,181): alarm colour if .goSTOP
button at (20,140)-(101,171): text "СТОП"; toggles .goSTOP
rounded rectangle at (10,70)-(111,121): alarm colour if .goPusk
button at (20,80)-(101,111): text "ПУСК"; toggles .goPusk
rounded rectangle at (10,10)-(111,61): alarm colour if .goRejim
button at (20,20)-(101,51): text "РЕЖИМ"; toggles .goRejim
*)
